FUNCTION_BLOCK FB_GuidanceSystem
VAR_INPUT
END_VAR
VAR_OUTPUT
	eCondition : eConditionCheck;
END_VAR
VAR
	fbAccelerationSensor1 : FB_AccelerationSensor;
	fbAccelerationSensor2 : FB_AccelerationSensor;
	
	eMode : eSystemMode;
END_VAR

CASE eMode OF
	eSystemMode.RUN :
		fbAccelerationSensor1();
		fbAccelerationSensor2();
		
		//Condition
		IF fbAccelerationSensor1.eCondition = eConditionCheck.INIT OR fbAccelerationSensor2.eCondition = eConditionCheck.INIT THEN
			eCondition := eConditionCheck.INIT;
		ELSIF fbAccelerationSensor1.eCondition = eConditionCheck.ERROR OR fbAccelerationSensor2.eCondition = eConditionCheck.ERROR THEN
			eCondition := eConditionCheck.ERROR;
		ELSIF fbAccelerationSensor1.eCondition = eConditionCheck.READY AND fbAccelerationSensor2.eCondition = eConditionCheck.READY THEN
			eCondition := eConditionCheck.READY;
		END_IF
			
	eSystemMode.SLEEP :
		//Condition
		eCondition := eConditionCheck.SLEEP;
END_CASE

PROPERTY getAccelerationSensor1 : ARRAY [0..2] OF REAL
GET
getAccelerationSensor1 := fbAccelerationSensor1.getAcceleration;
END_GET
END_PROPERTY

PROPERTY getAccelerationSensor2 : ARRAY [0..2] OF REAL
GET
getAccelerationSensor2 := fbAccelerationSensor1.getAcceleration;
END_GET
END_PROPERTY

PROPERTY setSLEEP : BOOL
SET
VAR
	e: INT;
END_VAR
IF setSLEEP THEN
	eMode := eSystemMode.SLEEP;
ELSE
	eMode := eSystemMode.RUN;
END_IF
END_SET
END_PROPERTY

END_FUNCTION_BLOCK

(* stored: Version 1.1.0.1, ProductVersion 3.1.4024.12
   POU FB_GuidanceSystem: Id {f33f1b41-c667-4ee8-81c9-ea9b824242db}, SpecialFunc None
   Property getAccelerationSensor1: Id {d02b525a-bc1b-492a-a816-47305250732e}
   Get Get: Id {a44a823d-8479-4c86-a9d4-e6594c5cc29d}
   Property getAccelerationSensor2: Id {77f151eb-f5be-47a3-8ffb-b31bed26cce9}
   Get Get: Id {dc8e6747-1f97-4ee1-9ae5-87cfe2fd9cb4}
   Property setSLEEP: Id {2c7bdcf5-f2be-4de0-8789-6ccbdaf498a7}
   Set Set: Id {adc99693-7db5-40c6-a798-c3aa93720eff} *)
